{attribute addProperty BoxType "EP2816-0008-0016"}
{attribute addProperty Id "Diag_InputAT %I*ARRAY[0 ..7] OF BOOL6480"}
{attribute addProperty CRC "265177097"}
{attribute addProperty SizeInBites "64"}
{attribute addProperty SizeInBytes "8"}
TYPE DO_Inputs_Channel_AC4A9AF0 :
STRUCT
	{attribute addProperty Name "Diag_Input"}
	Diag_Input AT %I* : ARRAY[0 ..7] OF BOOL;
END_STRUCT
END_TYPE

(* stored: Version 1.2.0.0, ProductVersion 3.1.4024.9
   DUT DO_Inputs_Channel_AC4A9AF0: Id {36d692e7-831a-4dee-bdc0-eecd27a1cb0a} *)
